// TIA Portal V19 export
FUNCTION "FC_001_Diagnostic" : Void   // FC12, LAD
{ S7_Optimized_Access := 'TRUE' }
// stored: SetENOAutomatically false
   VAR_IN_OUT
      Diagnostic7 : "DiagnosticMainCabinet";
      Diagnostic10 : "DiagnosticMainCabinet";
   END_VAR
BEGIN

REGION Network 1 (SCL)
   //************************************************************
   //===Author: Mateusz Połojko
   //-----Linkedin: https://pl.linkedin.com/in/mateusz-po%C5%82ojko-52a3541b1
   //-----Github: https://github.com/Bhazel95
   //===Description:
   //-----Diagnostic of hardware components
   //===Customer:
   //-----Apator Powogaz S.A.
   //************************************************************
END_REGION

REGION Network 2 (SCL)
   //Transporter 7A & 7B
   #Diagnostic7.ET_200SP.HeadModule_0.LADDR:= "IO_device_1~Head";
   #Diagnostic7.ET_200SP.HeadModule_0.Mode := 1;

   #Diagnostic7.ET_200SP.BusAdapter_1.LADDR := "IO_device_1~BusAdapter-Send_1xFC_1";
   #Diagnostic7.ET_200SP.BusAdapter_1.Mode := 1;

   #Diagnostic7.ET_200SP.InputSafety_2.LADDR := "IO_device_1~F-DI_8x24VDC_HF_1" ;
   #Diagnostic7.ET_200SP.InputSafety_2.Mode := 1;

   #Diagnostic7.ET_200SP.InputSafety_3.LADDR := "IO_device_1~F-DI_8x24VDC_HF_2";
   #Diagnostic7.ET_200SP.InputSafety_3.Mode := 1;

   #Diagnostic7.ET_200SP.InputSafety_4.LADDR := "IO_device_1~F-DI_8x24VDC_HF_3";
   #Diagnostic7.ET_200SP.InputSafety_4.Mode := 1;

   #Diagnostic7.ET_200SP.InputSafety_5.LADDR := "IO_device_1~F-DI_8x24VDC_HF_5";
   #Diagnostic7.ET_200SP.InputSafety_5.Mode := 1;

   #Diagnostic7.ET_200SP.InputSafety_6.LADDR := "IO_device_1~F-DI_8x24VDC_HF_4";
   #Diagnostic7.ET_200SP.InputSafety_6.Mode := 1;

   #Diagnostic7.ET_200SP.OutputSafety_7.LADDR := "IO_device_1~F-DQ_8x24VDC_0_5A_PP_HF_1";
   #Diagnostic7.ET_200SP.OutputSafety_7.Mode := 1;

   #Diagnostic7.ET_200SP.RelaySafety_9.LADDR := "IO_device_1~F-RQ_1x24__48VDC_24__230VAC_5A_1";
   #Diagnostic7.ET_200SP.RelaySafety_9.Mode := 1;

   #Diagnostic7.ET_200SP.RelaySafety_10.LADDR := "IO_device_1~F-RQ_1x24__48VDC_24__230VAC_5A_2";
   #Diagnostic7.ET_200SP.RelaySafety_10.Mode := 1;

   #Diagnostic7.ET_200SP.InputsDigital_11.LADDR := "IO_device_1~DI_16x24VDC_ST_1";
   #Diagnostic7.ET_200SP.InputsDigital_11.Mode := 1;

   #Diagnostic7.ET_200SP.InputsDigital_12.LADDR := "IO_device_1~DI_16x24VDC_ST_2";
   #Diagnostic7.ET_200SP.InputsDigital_12.Mode := 1;

   #Diagnostic7.ET_200SP.InputsDigital_13.LADDR := "IO_device_1~DI_16x24VDC_ST_3";
   #Diagnostic7.ET_200SP.InputsDigital_13.Mode := 1;

   #Diagnostic7.ET_200SP.InputAnalog_14.LADDR := "IO_device_1~AI_2xI_2-_4-wire_ST_1";
   #Diagnostic7.ET_200SP.InputAnalog_14.Mode := 1;

   #Diagnostic7.ET_200SP.OutputDigital_15.LADDR := "IO_device_1~DQ_16x24VDC_0_5A_ST_1";
   #Diagnostic7.ET_200SP.OutputDigital_15.Mode := 1;

   #Diagnostic7.ET_200SP.OutputDigital_16.LADDR := "IO_device_1~DQ_16x24VDC_0_5A_ST_2";
   #Diagnostic7.ET_200SP.OutputDigital_16.Mode := 1;

   #Diagnostic7.ET_200SP.OutputDigital_17.LADDR := "IO_device_1~DQ_16x24VDC_0_5A_ST_3";
   #Diagnostic7.ET_200SP.OutputDigital_17.Mode := 1;

   #Diagnostic7.ET_200SP.OutputDigital_18.LADDR := "IO_device_1~DQ_16x24VDC_0_5A_ST_4";
   #Diagnostic7.ET_200SP.OutputDigital_18.Mode := 1;

   #Diagnostic7.ET_200SP.OutputAnalog_19.LADDR := "IO_device_1~AQ_2xI_ST_1";
   #Diagnostic7.ET_200SP.OutputAnalog_19.Mode := 1;

   #Diagnostic7.ET_200SP.ET_200AL_1.LADDR := "IO_device_1~DI_8x24VDC_8xM8_1";
   #Diagnostic7.ET_200SP.ET_200AL_1.Mode := 1;

   #Diagnostic7.ET_200SP.ET_200AL_2.LADDR := "IO_device_1~DI_8x24VDC_8xM8_2";
   #Diagnostic7.ET_200SP.ET_200AL_2.Mode := 1;


   #Diagnostic7.SinamicG120_1.LADDR := "G120_CU250S_2_PN_VECTOR_7A~PROFINET_interface~IODevice";
   #Diagnostic7.SinamicG120_1.Mode := 1;

   #Diagnostic7.SinamicG120_1.LADDR := "G120_CU250S_2_PN_VECTOR_7B~PROFINET_interface~IODevice";
   #Diagnostic7.SinamicG120_1.Mode := 1;
END_REGION

REGION Network 3 (SCL)
   //Transporter 10A & 10B
   #Diagnostic10.ET_200SP.HeadModule_0.LADDR := "IO_device_2~Head";
   #Diagnostic10.ET_200SP.HeadModule_0.Mode := 1;

   #Diagnostic10.ET_200SP.BusAdapter_1.LADDR := "IO_device_2~BusAdapter-Send_1xFC_1";
   #Diagnostic10.ET_200SP.BusAdapter_1.Mode := 1;

   #Diagnostic10.ET_200SP.InputSafety_2.LADDR := "IO_device_2~F-DI_8x24VDC_HF_1";
   #Diagnostic10.ET_200SP.InputSafety_2.Mode := 1;

   #Diagnostic10.ET_200SP.InputSafety_3.LADDR := "IO_device_2~F-DI_8x24VDC_HF_2";
   #Diagnostic10.ET_200SP.InputSafety_3.Mode := 1;

   #Diagnostic10.ET_200SP.InputSafety_4.LADDR := "IO_device_2~F-DI_8x24VDC_HF_3";
   #Diagnostic10.ET_200SP.InputSafety_4.Mode := 1;

   #Diagnostic10.ET_200SP.InputSafety_5.LADDR := "IO_device_2~F-DI_8x24VDC_HF_4";
   #Diagnostic10.ET_200SP.InputSafety_5.Mode := 1;

   #Diagnostic10.ET_200SP.InputSafety_6.LADDR := "IO_device_2~F-DI_8x24VDC_HF_5";
   #Diagnostic10.ET_200SP.InputSafety_6.Mode := 1;

   #Diagnostic10.ET_200SP.OutputSafety_7.LADDR := "IO_device_2~F-DQ_8x24VDC_0_5A_PP_HF_1";
   #Diagnostic10.ET_200SP.OutputSafety_7.Mode := 1;

   #Diagnostic10.ET_200SP.RelaySafety_9.LADDR := "IO_device_2~F-RQ_1x24__48VDC_24__230VAC_5A_1";
   #Diagnostic10.ET_200SP.RelaySafety_9.Mode := 1;

   #Diagnostic10.ET_200SP.RelaySafety_10.LADDR := "IO_device_2~F-RQ_1x24__48VDC_24__230VAC_5A_2";
   #Diagnostic10.ET_200SP.RelaySafety_10.Mode := 1;

   #Diagnostic10.ET_200SP.InputsDigital_11.LADDR := "IO_device_2~DI_16x24VDC_ST_1";
   #Diagnostic10.ET_200SP.InputsDigital_11.Mode := 1;

   #Diagnostic10.ET_200SP.InputsDigital_12.LADDR := "IO_device_2~DI_16x24VDC_ST_2";
   #Diagnostic10.ET_200SP.InputsDigital_12.Mode := 1;

   #Diagnostic10.ET_200SP.InputsDigital_13.LADDR := "IO_device_2~DI_16x24VDC_ST_3";
   #Diagnostic10.ET_200SP.InputsDigital_13.Mode := 1;

   #Diagnostic10.ET_200SP.InputAnalog_14.LADDR := "IO_device_2~AI_2xI_2-_4-wire_ST_1";
   #Diagnostic10.ET_200SP.InputAnalog_14.Mode := 1;

   #Diagnostic10.ET_200SP.OutputDigital_15.LADDR := "IO_device_2~DQ_16x24VDC_0_5A_ST_1";
   #Diagnostic10.ET_200SP.OutputDigital_15.Mode := 1;

   #Diagnostic10.ET_200SP.OutputDigital_16.LADDR := "IO_device_2~DQ_16x24VDC_0_5A_ST_2";
   #Diagnostic10.ET_200SP.OutputDigital_16.Mode := 1;

   #Diagnostic10.ET_200SP.OutputDigital_17.LADDR := "IO_device_2~DQ_16x24VDC_0_5A_ST_3";
   #Diagnostic10.ET_200SP.OutputDigital_17.Mode := 1;

   #Diagnostic10.ET_200SP.OutputDigital_18.LADDR := "IO_device_2~DQ_16x24VDC_0_5A_ST_4";
   #Diagnostic10.ET_200SP.OutputDigital_18.Mode := 1;

   #Diagnostic10.ET_200SP.OutputAnalog_19.LADDR := "IO_device_2~AQ_2xI_ST_1";
   #Diagnostic10.ET_200SP.OutputAnalog_19.Mode := 1;

   #Diagnostic10.ET_200SP.ET_200AL_1.LADDR := "IO_device_2~DI_8x24VDC_8xM8_1";
   #Diagnostic10.ET_200SP.ET_200AL_1.Mode := 1;

   #Diagnostic10.ET_200SP.ET_200AL_2.LADDR := "IO_device_2~DI_8x24VDC_8xM8_2";
   #Diagnostic10.ET_200SP.ET_200AL_2.Mode := 1;


   #Diagnostic10.SinamicG120_1.LADDR := "G120_CU250S_2_PN_VECTOR_10A~PROFINET_interface~IODevice";
   #Diagnostic10.SinamicG120_1.Mode := 1;
END_REGION

REGION Network 4
   // ET 200SP - MODUL GLOWNY 7
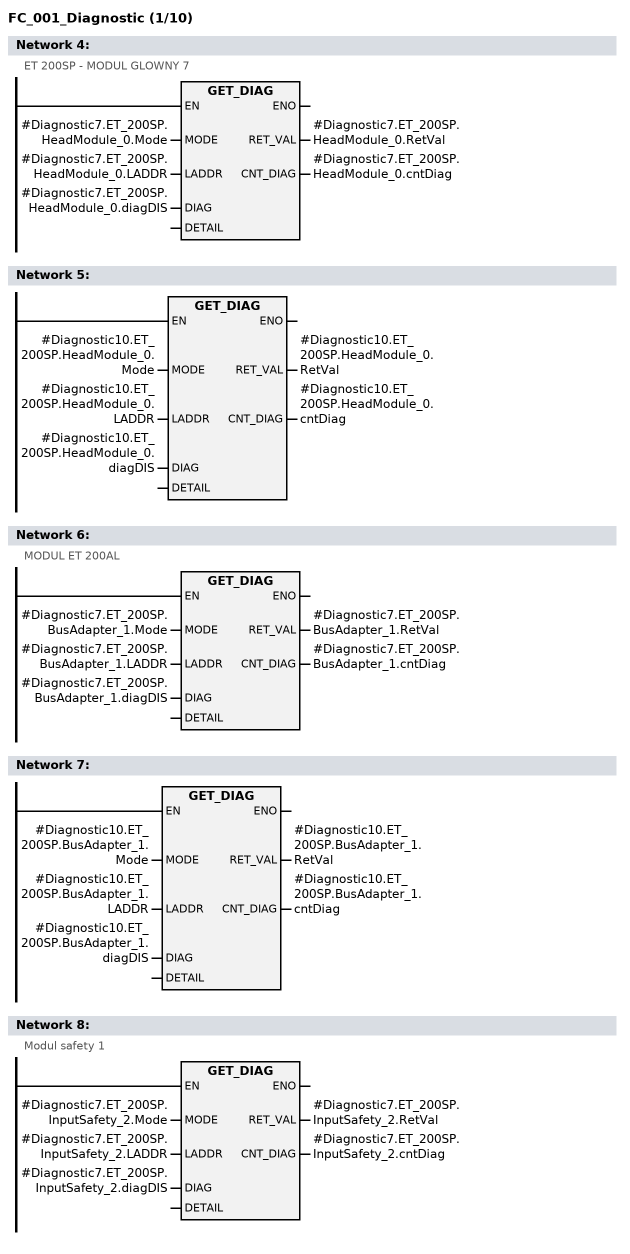
   RUNG wire#powerrail
      GET_DIAG(MODE := #Diagnostic7.ET_200SP.HeadModule_0.Mode, LADDR := #Diagnostic7.ET_200SP.HeadModule_0.LADDR, DIAG := #Diagnostic7.ET_200SP.HeadModule_0.diagDIS, DETAIL :=, RET_VAL => #Diagnostic7.ET_200SP.HeadModule_0.RetVal, CNT_DIAG => #Diagnostic7.ET_200SP.HeadModule_0.cntDiag)
   END_RUNG
   // the same network as SCL:
   #Diagnostic7.ET_200SP.HeadModule_0.RetVal := GET_DIAG(MODE := #Diagnostic7.ET_200SP.HeadModule_0.Mode,
                           LADDR := #Diagnostic7.ET_200SP.HeadModule_0.LADDR,
                           DIAG := #Diagnostic7.ET_200SP.HeadModule_0.diagDIS,
                           CNT_DIAG => #Diagnostic7.ET_200SP.HeadModule_0.cntDiag);
END_REGION

REGION Network 5
   RUNG wire#powerrail
      GET_DIAG(MODE := #Diagnostic10.ET_200SP.HeadModule_0.Mode, LADDR := #Diagnostic10.ET_200SP.HeadModule_0.LADDR, DIAG := #Diagnostic10.ET_200SP.HeadModule_0.diagDIS, DETAIL :=, RET_VAL => #Diagnostic10.ET_200SP.HeadModule_0.RetVal, CNT_DIAG => #Diagnostic10.ET_200SP.HeadModule_0.cntDiag)
   END_RUNG
   // the same network as SCL:
   #Diagnostic10.ET_200SP.HeadModule_0.RetVal := GET_DIAG(MODE := #Diagnostic10.ET_200SP.HeadModule_0.Mode,
                           LADDR := #Diagnostic10.ET_200SP.HeadModule_0.LADDR,
                           DIAG := #Diagnostic10.ET_200SP.HeadModule_0.diagDIS,
                           CNT_DIAG => #Diagnostic10.ET_200SP.HeadModule_0.cntDiag);
END_REGION

REGION Network 6
   // MODUL ET 200AL
   RUNG wire#powerrail
      GET_DIAG(MODE := #Diagnostic7.ET_200SP.BusAdapter_1.Mode, LADDR := #Diagnostic7.ET_200SP.BusAdapter_1.LADDR, DIAG := #Diagnostic7.ET_200SP.BusAdapter_1.diagDIS, DETAIL :=, RET_VAL => #Diagnostic7.ET_200SP.BusAdapter_1.RetVal, CNT_DIAG => #Diagnostic7.ET_200SP.BusAdapter_1.cntDiag)
   END_RUNG
   // the same network as SCL:
   #Diagnostic7.ET_200SP.BusAdapter_1.RetVal := GET_DIAG(MODE := #Diagnostic7.ET_200SP.BusAdapter_1.Mode,
                           LADDR := #Diagnostic7.ET_200SP.BusAdapter_1.LADDR,
                           DIAG := #Diagnostic7.ET_200SP.BusAdapter_1.diagDIS,
                           CNT_DIAG => #Diagnostic7.ET_200SP.BusAdapter_1.cntDiag);
END_REGION

REGION Network 7
   RUNG wire#powerrail
      GET_DIAG(MODE := #Diagnostic10.ET_200SP.BusAdapter_1.Mode, LADDR := #Diagnostic10.ET_200SP.BusAdapter_1.LADDR, DIAG := #Diagnostic10.ET_200SP.BusAdapter_1.diagDIS, DETAIL :=, RET_VAL => #Diagnostic10.ET_200SP.BusAdapter_1.RetVal, CNT_DIAG => #Diagnostic10.ET_200SP.BusAdapter_1.cntDiag)
   END_RUNG
   // the same network as SCL:
   #Diagnostic10.ET_200SP.BusAdapter_1.RetVal := GET_DIAG(MODE := #Diagnostic10.ET_200SP.BusAdapter_1.Mode,
                           LADDR := #Diagnostic10.ET_200SP.BusAdapter_1.LADDR,
                           DIAG := #Diagnostic10.ET_200SP.BusAdapter_1.diagDIS,
                           CNT_DIAG => #Diagnostic10.ET_200SP.BusAdapter_1.cntDiag);
END_REGION

REGION Network 8
   // Modul safety 1
   RUNG wire#powerrail
      GET_DIAG(MODE := #Diagnostic7.ET_200SP.InputSafety_2.Mode, LADDR := #Diagnostic7.ET_200SP.InputSafety_2.LADDR, DIAG := #Diagnostic7.ET_200SP.InputSafety_2.diagDIS, DETAIL :=, RET_VAL => #Diagnostic7.ET_200SP.InputSafety_2.RetVal, CNT_DIAG => #Diagnostic7.ET_200SP.InputSafety_2.cntDiag)
   END_RUNG
   // the same network as SCL:
   #Diagnostic7.ET_200SP.InputSafety_2.RetVal := GET_DIAG(MODE := #Diagnostic7.ET_200SP.InputSafety_2.Mode,
                           LADDR := #Diagnostic7.ET_200SP.InputSafety_2.LADDR,
                           DIAG := #Diagnostic7.ET_200SP.InputSafety_2.diagDIS,
                           CNT_DIAG => #Diagnostic7.ET_200SP.InputSafety_2.cntDiag);
END_REGION

REGION Network 9
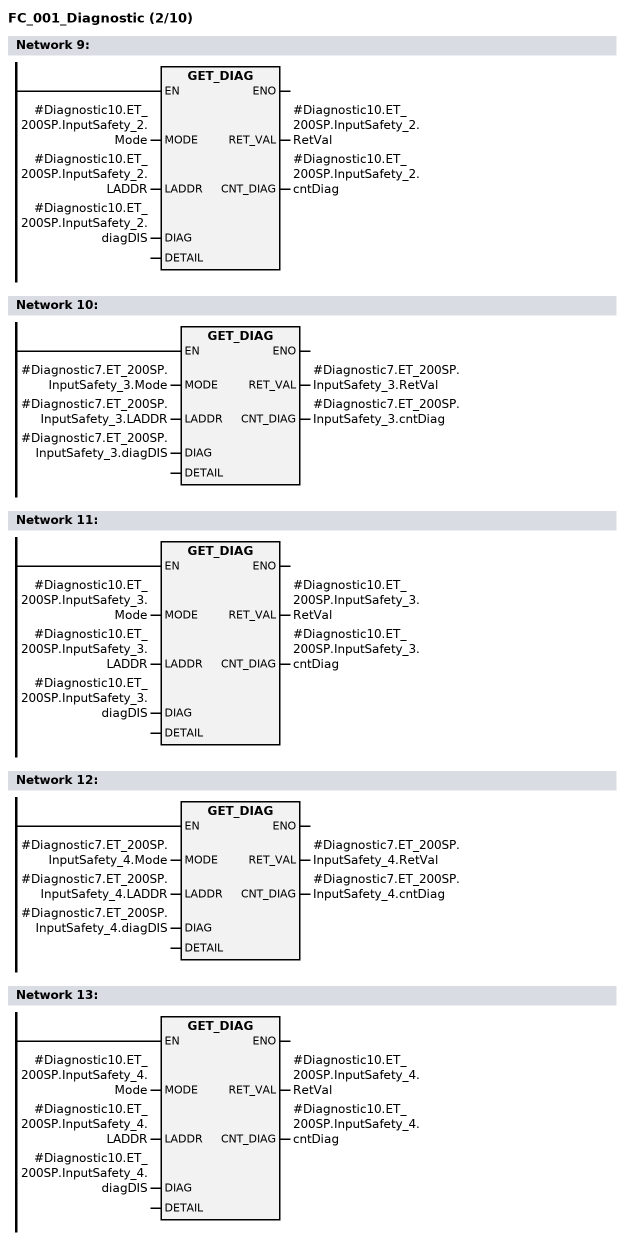
   RUNG wire#powerrail
      GET_DIAG(MODE := #Diagnostic10.ET_200SP.InputSafety_2.Mode, LADDR := #Diagnostic10.ET_200SP.InputSafety_2.LADDR, DIAG := #Diagnostic10.ET_200SP.InputSafety_2.diagDIS, DETAIL :=, RET_VAL => #Diagnostic10.ET_200SP.InputSafety_2.RetVal, CNT_DIAG => #Diagnostic10.ET_200SP.InputSafety_2.cntDiag)
   END_RUNG
   // the same network as SCL:
   #Diagnostic10.ET_200SP.InputSafety_2.RetVal := GET_DIAG(MODE := #Diagnostic10.ET_200SP.InputSafety_2.Mode,
                           LADDR := #Diagnostic10.ET_200SP.InputSafety_2.LADDR,
                           DIAG := #Diagnostic10.ET_200SP.InputSafety_2.diagDIS,
                           CNT_DIAG => #Diagnostic10.ET_200SP.InputSafety_2.cntDiag);
END_REGION

REGION Network 10
   RUNG wire#powerrail
      GET_DIAG(MODE := #Diagnostic7.ET_200SP.InputSafety_3.Mode, LADDR := #Diagnostic7.ET_200SP.InputSafety_3.LADDR, DIAG := #Diagnostic7.ET_200SP.InputSafety_3.diagDIS, DETAIL :=, RET_VAL => #Diagnostic7.ET_200SP.InputSafety_3.RetVal, CNT_DIAG => #Diagnostic7.ET_200SP.InputSafety_3.cntDiag)
   END_RUNG
   // the same network as SCL:
   #Diagnostic7.ET_200SP.InputSafety_3.RetVal := GET_DIAG(MODE := #Diagnostic7.ET_200SP.InputSafety_3.Mode,
                           LADDR := #Diagnostic7.ET_200SP.InputSafety_3.LADDR,
                           DIAG := #Diagnostic7.ET_200SP.InputSafety_3.diagDIS,
                           CNT_DIAG => #Diagnostic7.ET_200SP.InputSafety_3.cntDiag);
END_REGION

REGION Network 11
   RUNG wire#powerrail
      GET_DIAG(MODE := #Diagnostic10.ET_200SP.InputSafety_3.Mode, LADDR := #Diagnostic10.ET_200SP.InputSafety_3.LADDR, DIAG := #Diagnostic10.ET_200SP.InputSafety_3.diagDIS, DETAIL :=, RET_VAL => #Diagnostic10.ET_200SP.InputSafety_3.RetVal, CNT_DIAG => #Diagnostic10.ET_200SP.InputSafety_3.cntDiag)
   END_RUNG
   // the same network as SCL:
   #Diagnostic10.ET_200SP.InputSafety_3.RetVal := GET_DIAG(MODE := #Diagnostic10.ET_200SP.InputSafety_3.Mode,
                           LADDR := #Diagnostic10.ET_200SP.InputSafety_3.LADDR,
                           DIAG := #Diagnostic10.ET_200SP.InputSafety_3.diagDIS,
                           CNT_DIAG => #Diagnostic10.ET_200SP.InputSafety_3.cntDiag);
END_REGION

REGION Network 12
   RUNG wire#powerrail
      GET_DIAG(MODE := #Diagnostic7.ET_200SP.InputSafety_4.Mode, LADDR := #Diagnostic7.ET_200SP.InputSafety_4.LADDR, DIAG := #Diagnostic7.ET_200SP.InputSafety_4.diagDIS, DETAIL :=, RET_VAL => #Diagnostic7.ET_200SP.InputSafety_4.RetVal, CNT_DIAG => #Diagnostic7.ET_200SP.InputSafety_4.cntDiag)
   END_RUNG
   // the same network as SCL:
   #Diagnostic7.ET_200SP.InputSafety_4.RetVal := GET_DIAG(MODE := #Diagnostic7.ET_200SP.InputSafety_4.Mode,
                           LADDR := #Diagnostic7.ET_200SP.InputSafety_4.LADDR,
                           DIAG := #Diagnostic7.ET_200SP.InputSafety_4.diagDIS,
                           CNT_DIAG => #Diagnostic7.ET_200SP.InputSafety_4.cntDiag);
END_REGION

REGION Network 13
   RUNG wire#powerrail
      GET_DIAG(MODE := #Diagnostic10.ET_200SP.InputSafety_4.Mode, LADDR := #Diagnostic10.ET_200SP.InputSafety_4.LADDR, DIAG := #Diagnostic10.ET_200SP.InputSafety_4.diagDIS, DETAIL :=, RET_VAL => #Diagnostic10.ET_200SP.InputSafety_4.RetVal, CNT_DIAG => #Diagnostic10.ET_200SP.InputSafety_4.cntDiag)
   END_RUNG
   // the same network as SCL:
   #Diagnostic10.ET_200SP.InputSafety_4.RetVal := GET_DIAG(MODE := #Diagnostic10.ET_200SP.InputSafety_4.Mode,
                           LADDR := #Diagnostic10.ET_200SP.InputSafety_4.LADDR,
                           DIAG := #Diagnostic10.ET_200SP.InputSafety_4.diagDIS,
                           CNT_DIAG => #Diagnostic10.ET_200SP.InputSafety_4.cntDiag);
END_REGION

REGION Network 14
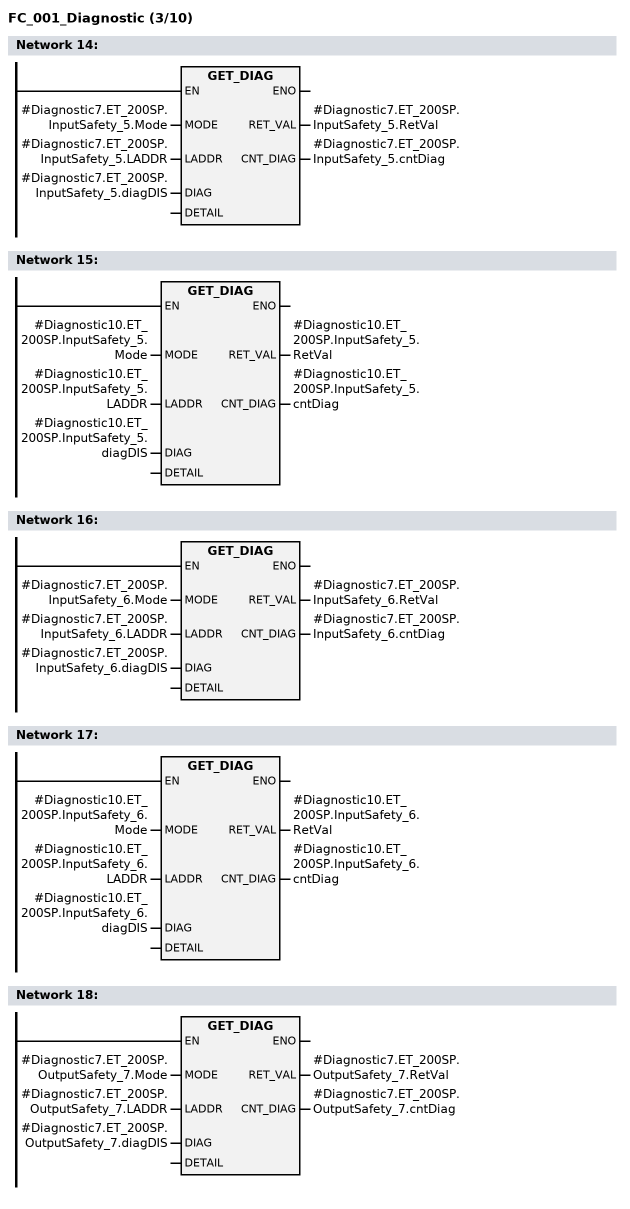
   RUNG wire#powerrail
      GET_DIAG(MODE := #Diagnostic7.ET_200SP.InputSafety_5.Mode, LADDR := #Diagnostic7.ET_200SP.InputSafety_5.LADDR, DIAG := #Diagnostic7.ET_200SP.InputSafety_5.diagDIS, DETAIL :=, RET_VAL => #Diagnostic7.ET_200SP.InputSafety_5.RetVal, CNT_DIAG => #Diagnostic7.ET_200SP.InputSafety_5.cntDiag)
   END_RUNG
   // the same network as SCL:
   #Diagnostic7.ET_200SP.InputSafety_5.RetVal := GET_DIAG(MODE := #Diagnostic7.ET_200SP.InputSafety_5.Mode,
                           LADDR := #Diagnostic7.ET_200SP.InputSafety_5.LADDR,
                           DIAG := #Diagnostic7.ET_200SP.InputSafety_5.diagDIS,
                           CNT_DIAG => #Diagnostic7.ET_200SP.InputSafety_5.cntDiag);
END_REGION

REGION Network 15
   RUNG wire#powerrail
      GET_DIAG(MODE := #Diagnostic10.ET_200SP.InputSafety_5.Mode, LADDR := #Diagnostic10.ET_200SP.InputSafety_5.LADDR, DIAG := #Diagnostic10.ET_200SP.InputSafety_5.diagDIS, DETAIL :=, RET_VAL => #Diagnostic10.ET_200SP.InputSafety_5.RetVal, CNT_DIAG => #Diagnostic10.ET_200SP.InputSafety_5.cntDiag)
   END_RUNG
   // the same network as SCL:
   #Diagnostic10.ET_200SP.InputSafety_5.RetVal := GET_DIAG(MODE := #Diagnostic10.ET_200SP.InputSafety_5.Mode,
                           LADDR := #Diagnostic10.ET_200SP.InputSafety_5.LADDR,
                           DIAG := #Diagnostic10.ET_200SP.InputSafety_5.diagDIS,
                           CNT_DIAG => #Diagnostic10.ET_200SP.InputSafety_5.cntDiag);
END_REGION

REGION Network 16
   RUNG wire#powerrail
      GET_DIAG(MODE := #Diagnostic7.ET_200SP.InputSafety_6.Mode, LADDR := #Diagnostic7.ET_200SP.InputSafety_6.LADDR, DIAG := #Diagnostic7.ET_200SP.InputSafety_6.diagDIS, DETAIL :=, RET_VAL => #Diagnostic7.ET_200SP.InputSafety_6.RetVal, CNT_DIAG => #Diagnostic7.ET_200SP.InputSafety_6.cntDiag)
   END_RUNG
   // the same network as SCL:
   #Diagnostic7.ET_200SP.InputSafety_6.RetVal := GET_DIAG(MODE := #Diagnostic7.ET_200SP.InputSafety_6.Mode,
                           LADDR := #Diagnostic7.ET_200SP.InputSafety_6.LADDR,
                           DIAG := #Diagnostic7.ET_200SP.InputSafety_6.diagDIS,
                           CNT_DIAG => #Diagnostic7.ET_200SP.InputSafety_6.cntDiag);
END_REGION

REGION Network 17
   RUNG wire#powerrail
      GET_DIAG(MODE := #Diagnostic10.ET_200SP.InputSafety_6.Mode, LADDR := #Diagnostic10.ET_200SP.InputSafety_6.LADDR, DIAG := #Diagnostic10.ET_200SP.InputSafety_6.diagDIS, DETAIL :=, RET_VAL => #Diagnostic10.ET_200SP.InputSafety_6.RetVal, CNT_DIAG => #Diagnostic10.ET_200SP.InputSafety_6.cntDiag)
   END_RUNG
   // the same network as SCL:
   #Diagnostic10.ET_200SP.InputSafety_6.RetVal := GET_DIAG(MODE := #Diagnostic10.ET_200SP.InputSafety_6.Mode,
                           LADDR := #Diagnostic10.ET_200SP.InputSafety_6.LADDR,
                           DIAG := #Diagnostic10.ET_200SP.InputSafety_6.diagDIS,
                           CNT_DIAG => #Diagnostic10.ET_200SP.InputSafety_6.cntDiag);
END_REGION

REGION Network 18
   RUNG wire#powerrail
      GET_DIAG(MODE := #Diagnostic7.ET_200SP.OutputSafety_7.Mode, LADDR := #Diagnostic7.ET_200SP.OutputSafety_7.LADDR, DIAG := #Diagnostic7.ET_200SP.OutputSafety_7.diagDIS, DETAIL :=, RET_VAL => #Diagnostic7.ET_200SP.OutputSafety_7.RetVal, CNT_DIAG => #Diagnostic7.ET_200SP.OutputSafety_7.cntDiag)
   END_RUNG
   // the same network as SCL:
   #Diagnostic7.ET_200SP.OutputSafety_7.RetVal := GET_DIAG(MODE := #Diagnostic7.ET_200SP.OutputSafety_7.Mode,
                           LADDR := #Diagnostic7.ET_200SP.OutputSafety_7.LADDR,
                           DIAG := #Diagnostic7.ET_200SP.OutputSafety_7.diagDIS,
                           CNT_DIAG => #Diagnostic7.ET_200SP.OutputSafety_7.cntDiag);
END_REGION

REGION Network 19
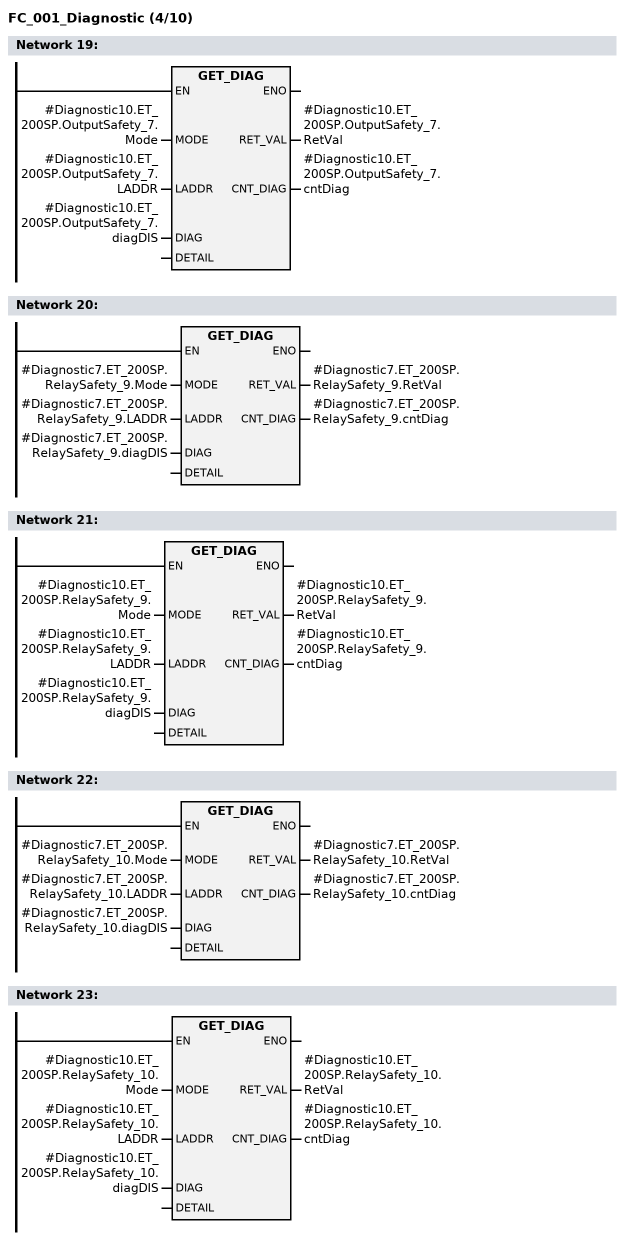
   RUNG wire#powerrail
      GET_DIAG(MODE := #Diagnostic10.ET_200SP.OutputSafety_7.Mode, LADDR := #Diagnostic10.ET_200SP.OutputSafety_7.LADDR, DIAG := #Diagnostic10.ET_200SP.OutputSafety_7.diagDIS, DETAIL :=, RET_VAL => #Diagnostic10.ET_200SP.OutputSafety_7.RetVal, CNT_DIAG => #Diagnostic10.ET_200SP.OutputSafety_7.cntDiag)
   END_RUNG
   // the same network as SCL:
   #Diagnostic10.ET_200SP.OutputSafety_7.RetVal := GET_DIAG(MODE := #Diagnostic10.ET_200SP.OutputSafety_7.Mode,
                           LADDR := #Diagnostic10.ET_200SP.OutputSafety_7.LADDR,
                           DIAG := #Diagnostic10.ET_200SP.OutputSafety_7.diagDIS,
                           CNT_DIAG => #Diagnostic10.ET_200SP.OutputSafety_7.cntDiag);
END_REGION

REGION Network 20
   RUNG wire#powerrail
      GET_DIAG(MODE := #Diagnostic7.ET_200SP.RelaySafety_9.Mode, LADDR := #Diagnostic7.ET_200SP.RelaySafety_9.LADDR, DIAG := #Diagnostic7.ET_200SP.RelaySafety_9.diagDIS, DETAIL :=, RET_VAL => #Diagnostic7.ET_200SP.RelaySafety_9.RetVal, CNT_DIAG => #Diagnostic7.ET_200SP.RelaySafety_9.cntDiag)
   END_RUNG
   // the same network as SCL:
   #Diagnostic7.ET_200SP.RelaySafety_9.RetVal := GET_DIAG(MODE := #Diagnostic7.ET_200SP.RelaySafety_9.Mode,
                           LADDR := #Diagnostic7.ET_200SP.RelaySafety_9.LADDR,
                           DIAG := #Diagnostic7.ET_200SP.RelaySafety_9.diagDIS,
                           CNT_DIAG => #Diagnostic7.ET_200SP.RelaySafety_9.cntDiag);
END_REGION

REGION Network 21
   RUNG wire#powerrail
      GET_DIAG(MODE := #Diagnostic10.ET_200SP.RelaySafety_9.Mode, LADDR := #Diagnostic10.ET_200SP.RelaySafety_9.LADDR, DIAG := #Diagnostic10.ET_200SP.RelaySafety_9.diagDIS, DETAIL :=, RET_VAL => #Diagnostic10.ET_200SP.RelaySafety_9.RetVal, CNT_DIAG => #Diagnostic10.ET_200SP.RelaySafety_9.cntDiag)
   END_RUNG
   // the same network as SCL:
   #Diagnostic10.ET_200SP.RelaySafety_9.RetVal := GET_DIAG(MODE := #Diagnostic10.ET_200SP.RelaySafety_9.Mode,
                           LADDR := #Diagnostic10.ET_200SP.RelaySafety_9.LADDR,
                           DIAG := #Diagnostic10.ET_200SP.RelaySafety_9.diagDIS,
                           CNT_DIAG => #Diagnostic10.ET_200SP.RelaySafety_9.cntDiag);
END_REGION

REGION Network 22
   RUNG wire#powerrail
      GET_DIAG(MODE := #Diagnostic7.ET_200SP.RelaySafety_10.Mode, LADDR := #Diagnostic7.ET_200SP.RelaySafety_10.LADDR, DIAG := #Diagnostic7.ET_200SP.RelaySafety_10.diagDIS, DETAIL :=, RET_VAL => #Diagnostic7.ET_200SP.RelaySafety_10.RetVal, CNT_DIAG => #Diagnostic7.ET_200SP.RelaySafety_10.cntDiag)
   END_RUNG
   // the same network as SCL:
   #Diagnostic7.ET_200SP.RelaySafety_10.RetVal := GET_DIAG(MODE := #Diagnostic7.ET_200SP.RelaySafety_10.Mode,
                           LADDR := #Diagnostic7.ET_200SP.RelaySafety_10.LADDR,
                           DIAG := #Diagnostic7.ET_200SP.RelaySafety_10.diagDIS,
                           CNT_DIAG => #Diagnostic7.ET_200SP.RelaySafety_10.cntDiag);
END_REGION

REGION Network 23
   RUNG wire#powerrail
      GET_DIAG(MODE := #Diagnostic10.ET_200SP.RelaySafety_10.Mode, LADDR := #Diagnostic10.ET_200SP.RelaySafety_10.LADDR, DIAG := #Diagnostic10.ET_200SP.RelaySafety_10.diagDIS, DETAIL :=, RET_VAL => #Diagnostic10.ET_200SP.RelaySafety_10.RetVal, CNT_DIAG => #Diagnostic10.ET_200SP.RelaySafety_10.cntDiag)
   END_RUNG
   // the same network as SCL:
   #Diagnostic10.ET_200SP.RelaySafety_10.RetVal := GET_DIAG(MODE := #Diagnostic10.ET_200SP.RelaySafety_10.Mode,
                           LADDR := #Diagnostic10.ET_200SP.RelaySafety_10.LADDR,
                           DIAG := #Diagnostic10.ET_200SP.RelaySafety_10.diagDIS,
                           CNT_DIAG => #Diagnostic10.ET_200SP.RelaySafety_10.cntDiag);
END_REGION

REGION Network 24
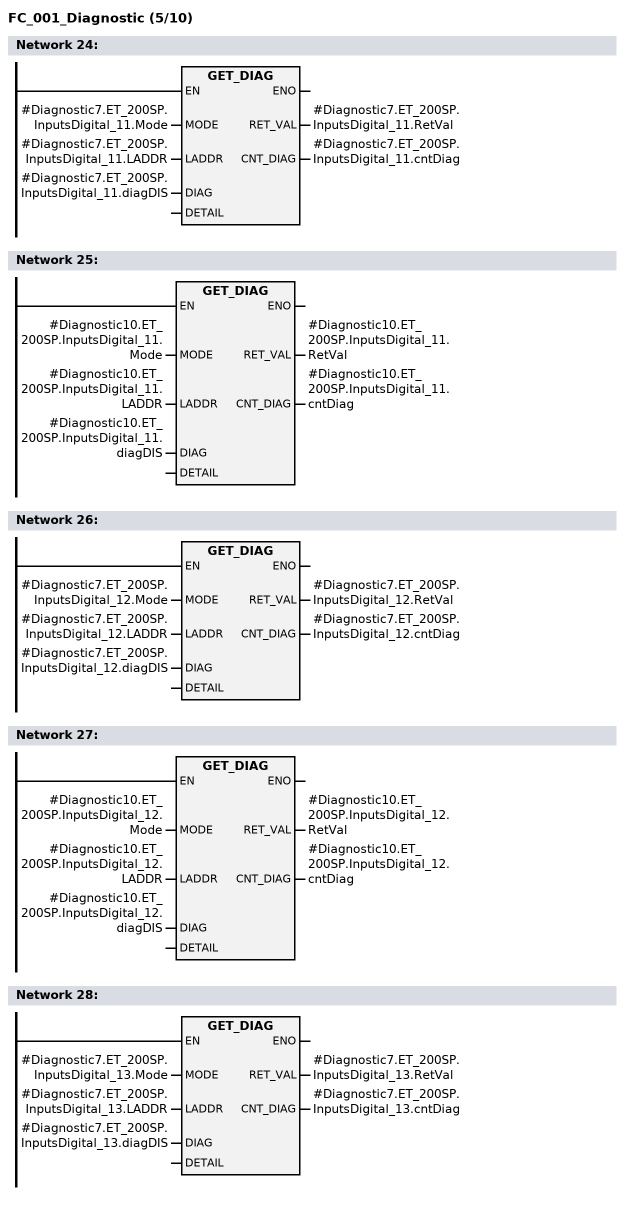
   RUNG wire#powerrail
      GET_DIAG(MODE := #Diagnostic7.ET_200SP.InputsDigital_11.Mode, LADDR := #Diagnostic7.ET_200SP.InputsDigital_11.LADDR, DIAG := #Diagnostic7.ET_200SP.InputsDigital_11.diagDIS, DETAIL :=, RET_VAL => #Diagnostic7.ET_200SP.InputsDigital_11.RetVal, CNT_DIAG => #Diagnostic7.ET_200SP.InputsDigital_11.cntDiag)
   END_RUNG
   // the same network as SCL:
   #Diagnostic7.ET_200SP.InputsDigital_11.RetVal := GET_DIAG(MODE := #Diagnostic7.ET_200SP.InputsDigital_11.Mode,
                           LADDR := #Diagnostic7.ET_200SP.InputsDigital_11.LADDR,
                           DIAG := #Diagnostic7.ET_200SP.InputsDigital_11.diagDIS,
                           CNT_DIAG => #Diagnostic7.ET_200SP.InputsDigital_11.cntDiag);
END_REGION

REGION Network 25
   RUNG wire#powerrail
      GET_DIAG(MODE := #Diagnostic10.ET_200SP.InputsDigital_11.Mode, LADDR := #Diagnostic10.ET_200SP.InputsDigital_11.LADDR, DIAG := #Diagnostic10.ET_200SP.InputsDigital_11.diagDIS, DETAIL :=, RET_VAL => #Diagnostic10.ET_200SP.InputsDigital_11.RetVal, CNT_DIAG => #Diagnostic10.ET_200SP.InputsDigital_11.cntDiag)
   END_RUNG
   // the same network as SCL:
   #Diagnostic10.ET_200SP.InputsDigital_11.RetVal := GET_DIAG(MODE := #Diagnostic10.ET_200SP.InputsDigital_11.Mode,
                           LADDR := #Diagnostic10.ET_200SP.InputsDigital_11.LADDR,
                           DIAG := #Diagnostic10.ET_200SP.InputsDigital_11.diagDIS,
                           CNT_DIAG => #Diagnostic10.ET_200SP.InputsDigital_11.cntDiag);
END_REGION

REGION Network 26
   RUNG wire#powerrail
      GET_DIAG(MODE := #Diagnostic7.ET_200SP.InputsDigital_12.Mode, LADDR := #Diagnostic7.ET_200SP.InputsDigital_12.LADDR, DIAG := #Diagnostic7.ET_200SP.InputsDigital_12.diagDIS, DETAIL :=, RET_VAL => #Diagnostic7.ET_200SP.InputsDigital_12.RetVal, CNT_DIAG => #Diagnostic7.ET_200SP.InputsDigital_12.cntDiag)
   END_RUNG
   // the same network as SCL:
   #Diagnostic7.ET_200SP.InputsDigital_12.RetVal := GET_DIAG(MODE := #Diagnostic7.ET_200SP.InputsDigital_12.Mode,
                           LADDR := #Diagnostic7.ET_200SP.InputsDigital_12.LADDR,
                           DIAG := #Diagnostic7.ET_200SP.InputsDigital_12.diagDIS,
                           CNT_DIAG => #Diagnostic7.ET_200SP.InputsDigital_12.cntDiag);
END_REGION

REGION Network 27
   RUNG wire#powerrail
      GET_DIAG(MODE := #Diagnostic10.ET_200SP.InputsDigital_12.Mode, LADDR := #Diagnostic10.ET_200SP.InputsDigital_12.LADDR, DIAG := #Diagnostic10.ET_200SP.InputsDigital_12.diagDIS, DETAIL :=, RET_VAL => #Diagnostic10.ET_200SP.InputsDigital_12.RetVal, CNT_DIAG => #Diagnostic10.ET_200SP.InputsDigital_12.cntDiag)
   END_RUNG
   // the same network as SCL:
   #Diagnostic10.ET_200SP.InputsDigital_12.RetVal := GET_DIAG(MODE := #Diagnostic10.ET_200SP.InputsDigital_12.Mode,
                           LADDR := #Diagnostic10.ET_200SP.InputsDigital_12.LADDR,
                           DIAG := #Diagnostic10.ET_200SP.InputsDigital_12.diagDIS,
                           CNT_DIAG => #Diagnostic10.ET_200SP.InputsDigital_12.cntDiag);
END_REGION

REGION Network 28
   RUNG wire#powerrail
      GET_DIAG(MODE := #Diagnostic7.ET_200SP.InputsDigital_13.Mode, LADDR := #Diagnostic7.ET_200SP.InputsDigital_13.LADDR, DIAG := #Diagnostic7.ET_200SP.InputsDigital_13.diagDIS, DETAIL :=, RET_VAL => #Diagnostic7.ET_200SP.InputsDigital_13.RetVal, CNT_DIAG => #Diagnostic7.ET_200SP.InputsDigital_13.cntDiag)
   END_RUNG
   // the same network as SCL:
   #Diagnostic7.ET_200SP.InputsDigital_13.RetVal := GET_DIAG(MODE := #Diagnostic7.ET_200SP.InputsDigital_13.Mode,
                           LADDR := #Diagnostic7.ET_200SP.InputsDigital_13.LADDR,
                           DIAG := #Diagnostic7.ET_200SP.InputsDigital_13.diagDIS,
                           CNT_DIAG => #Diagnostic7.ET_200SP.InputsDigital_13.cntDiag);
END_REGION

REGION Network 29
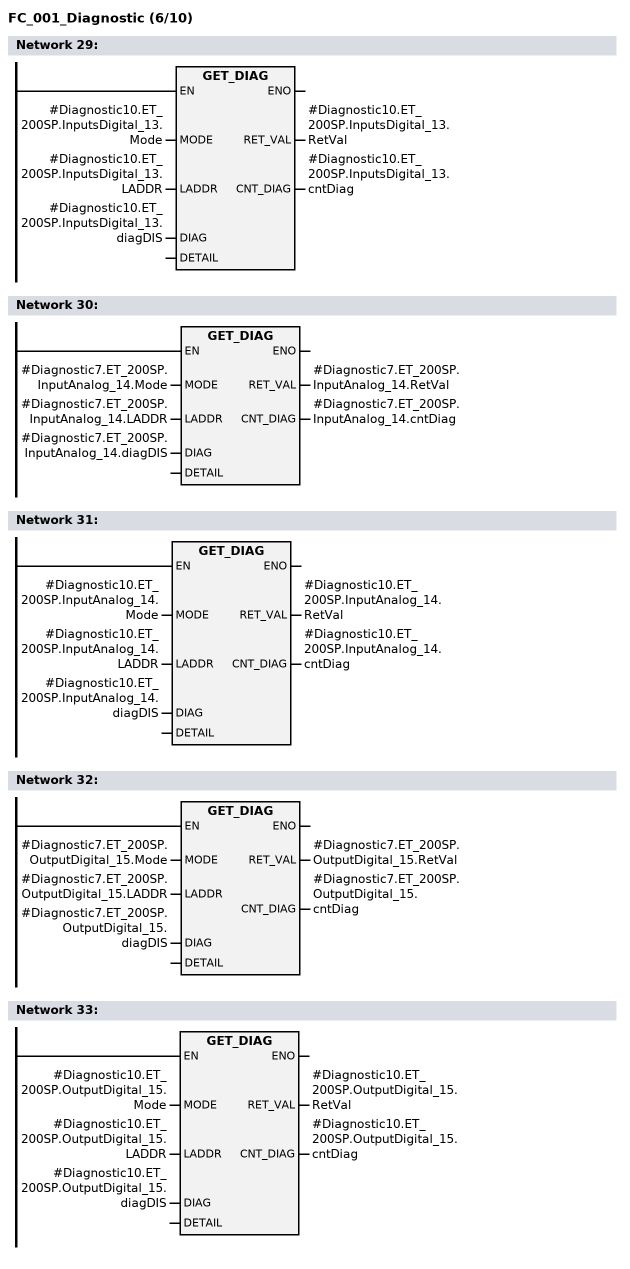
   RUNG wire#powerrail
      GET_DIAG(MODE := #Diagnostic10.ET_200SP.InputsDigital_13.Mode, LADDR := #Diagnostic10.ET_200SP.InputsDigital_13.LADDR, DIAG := #Diagnostic10.ET_200SP.InputsDigital_13.diagDIS, DETAIL :=, RET_VAL => #Diagnostic10.ET_200SP.InputsDigital_13.RetVal, CNT_DIAG => #Diagnostic10.ET_200SP.InputsDigital_13.cntDiag)
   END_RUNG
   // the same network as SCL:
   #Diagnostic10.ET_200SP.InputsDigital_13.RetVal := GET_DIAG(MODE := #Diagnostic10.ET_200SP.InputsDigital_13.Mode,
                           LADDR := #Diagnostic10.ET_200SP.InputsDigital_13.LADDR,
                           DIAG := #Diagnostic10.ET_200SP.InputsDigital_13.diagDIS,
                           CNT_DIAG => #Diagnostic10.ET_200SP.InputsDigital_13.cntDiag);
END_REGION

REGION Network 30
   RUNG wire#powerrail
      GET_DIAG(MODE := #Diagnostic7.ET_200SP.InputAnalog_14.Mode, LADDR := #Diagnostic7.ET_200SP.InputAnalog_14.LADDR, DIAG := #Diagnostic7.ET_200SP.InputAnalog_14.diagDIS, DETAIL :=, RET_VAL => #Diagnostic7.ET_200SP.InputAnalog_14.RetVal, CNT_DIAG => #Diagnostic7.ET_200SP.InputAnalog_14.cntDiag)
   END_RUNG
   // the same network as SCL:
   #Diagnostic7.ET_200SP.InputAnalog_14.RetVal := GET_DIAG(MODE := #Diagnostic7.ET_200SP.InputAnalog_14.Mode,
                           LADDR := #Diagnostic7.ET_200SP.InputAnalog_14.LADDR,
                           DIAG := #Diagnostic7.ET_200SP.InputAnalog_14.diagDIS,
                           CNT_DIAG => #Diagnostic7.ET_200SP.InputAnalog_14.cntDiag);
END_REGION

REGION Network 31
   RUNG wire#powerrail
      GET_DIAG(MODE := #Diagnostic10.ET_200SP.InputAnalog_14.Mode, LADDR := #Diagnostic10.ET_200SP.InputAnalog_14.LADDR, DIAG := #Diagnostic10.ET_200SP.InputAnalog_14.diagDIS, DETAIL :=, RET_VAL => #Diagnostic10.ET_200SP.InputAnalog_14.RetVal, CNT_DIAG => #Diagnostic10.ET_200SP.InputAnalog_14.cntDiag)
   END_RUNG
   // the same network as SCL:
   #Diagnostic10.ET_200SP.InputAnalog_14.RetVal := GET_DIAG(MODE := #Diagnostic10.ET_200SP.InputAnalog_14.Mode,
                           LADDR := #Diagnostic10.ET_200SP.InputAnalog_14.LADDR,
                           DIAG := #Diagnostic10.ET_200SP.InputAnalog_14.diagDIS,
                           CNT_DIAG => #Diagnostic10.ET_200SP.InputAnalog_14.cntDiag);
END_REGION

REGION Network 32
   RUNG wire#powerrail
      GET_DIAG(MODE := #Diagnostic7.ET_200SP.OutputDigital_15.Mode, LADDR := #Diagnostic7.ET_200SP.OutputDigital_15.LADDR, DIAG := #Diagnostic7.ET_200SP.OutputDigital_15.diagDIS, DETAIL :=, RET_VAL => #Diagnostic7.ET_200SP.OutputDigital_15.RetVal, CNT_DIAG => #Diagnostic7.ET_200SP.OutputDigital_15.cntDiag)
   END_RUNG
   // the same network as SCL:
   #Diagnostic7.ET_200SP.OutputDigital_15.RetVal := GET_DIAG(MODE := #Diagnostic7.ET_200SP.OutputDigital_15.Mode,
                           LADDR := #Diagnostic7.ET_200SP.OutputDigital_15.LADDR,
                           DIAG := #Diagnostic7.ET_200SP.OutputDigital_15.diagDIS,
                           CNT_DIAG => #Diagnostic7.ET_200SP.OutputDigital_15.cntDiag);
END_REGION

REGION Network 33
   RUNG wire#powerrail
      GET_DIAG(MODE := #Diagnostic10.ET_200SP.OutputDigital_15.Mode, LADDR := #Diagnostic10.ET_200SP.OutputDigital_15.LADDR, DIAG := #Diagnostic10.ET_200SP.OutputDigital_15.diagDIS, DETAIL :=, RET_VAL => #Diagnostic10.ET_200SP.OutputDigital_15.RetVal, CNT_DIAG => #Diagnostic10.ET_200SP.OutputDigital_15.cntDiag)
   END_RUNG
   // the same network as SCL:
   #Diagnostic10.ET_200SP.OutputDigital_15.RetVal := GET_DIAG(MODE := #Diagnostic10.ET_200SP.OutputDigital_15.Mode,
                           LADDR := #Diagnostic10.ET_200SP.OutputDigital_15.LADDR,
                           DIAG := #Diagnostic10.ET_200SP.OutputDigital_15.diagDIS,
                           CNT_DIAG => #Diagnostic10.ET_200SP.OutputDigital_15.cntDiag);
END_REGION

REGION Network 34
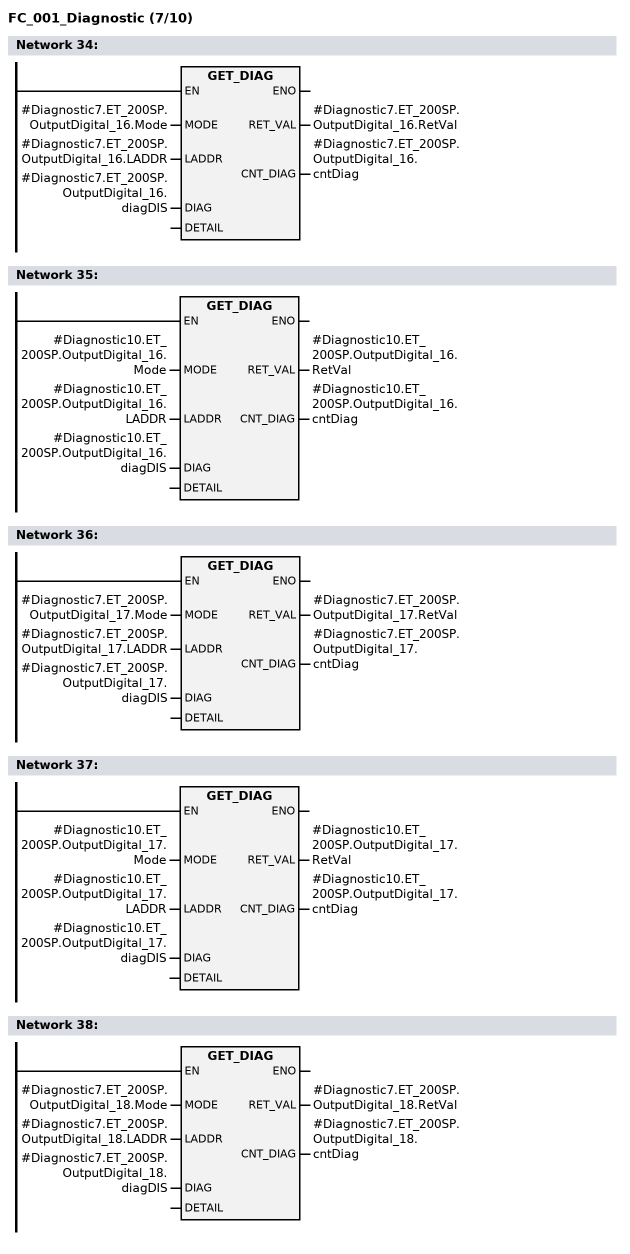
   RUNG wire#powerrail
      GET_DIAG(MODE := #Diagnostic7.ET_200SP.OutputDigital_16.Mode, LADDR := #Diagnostic7.ET_200SP.OutputDigital_16.LADDR, DIAG := #Diagnostic7.ET_200SP.OutputDigital_16.diagDIS, DETAIL :=, RET_VAL => #Diagnostic7.ET_200SP.OutputDigital_16.RetVal, CNT_DIAG => #Diagnostic7.ET_200SP.OutputDigital_16.cntDiag)
   END_RUNG
   // the same network as SCL:
   #Diagnostic7.ET_200SP.OutputDigital_16.RetVal := GET_DIAG(MODE := #Diagnostic7.ET_200SP.OutputDigital_16.Mode,
                           LADDR := #Diagnostic7.ET_200SP.OutputDigital_16.LADDR,
                           DIAG := #Diagnostic7.ET_200SP.OutputDigital_16.diagDIS,
                           CNT_DIAG => #Diagnostic7.ET_200SP.OutputDigital_16.cntDiag);
END_REGION

REGION Network 35
   RUNG wire#powerrail
      GET_DIAG(MODE := #Diagnostic10.ET_200SP.OutputDigital_16.Mode, LADDR := #Diagnostic10.ET_200SP.OutputDigital_16.LADDR, DIAG := #Diagnostic10.ET_200SP.OutputDigital_16.diagDIS, DETAIL :=, RET_VAL => #Diagnostic10.ET_200SP.OutputDigital_16.RetVal, CNT_DIAG => #Diagnostic10.ET_200SP.OutputDigital_16.cntDiag)
   END_RUNG
   // the same network as SCL:
   #Diagnostic10.ET_200SP.OutputDigital_16.RetVal := GET_DIAG(MODE := #Diagnostic10.ET_200SP.OutputDigital_16.Mode,
                           LADDR := #Diagnostic10.ET_200SP.OutputDigital_16.LADDR,
                           DIAG := #Diagnostic10.ET_200SP.OutputDigital_16.diagDIS,
                           CNT_DIAG => #Diagnostic10.ET_200SP.OutputDigital_16.cntDiag);
END_REGION

REGION Network 36
   RUNG wire#powerrail
      GET_DIAG(MODE := #Diagnostic7.ET_200SP.OutputDigital_17.Mode, LADDR := #Diagnostic7.ET_200SP.OutputDigital_17.LADDR, DIAG := #Diagnostic7.ET_200SP.OutputDigital_17.diagDIS, DETAIL :=, RET_VAL => #Diagnostic7.ET_200SP.OutputDigital_17.RetVal, CNT_DIAG => #Diagnostic7.ET_200SP.OutputDigital_17.cntDiag)
   END_RUNG
   // the same network as SCL:
   #Diagnostic7.ET_200SP.OutputDigital_17.RetVal := GET_DIAG(MODE := #Diagnostic7.ET_200SP.OutputDigital_17.Mode,
                           LADDR := #Diagnostic7.ET_200SP.OutputDigital_17.LADDR,
                           DIAG := #Diagnostic7.ET_200SP.OutputDigital_17.diagDIS,
                           CNT_DIAG => #Diagnostic7.ET_200SP.OutputDigital_17.cntDiag);
END_REGION

REGION Network 37
   RUNG wire#powerrail
      GET_DIAG(MODE := #Diagnostic10.ET_200SP.OutputDigital_17.Mode, LADDR := #Diagnostic10.ET_200SP.OutputDigital_17.LADDR, DIAG := #Diagnostic10.ET_200SP.OutputDigital_17.diagDIS, DETAIL :=, RET_VAL => #Diagnostic10.ET_200SP.OutputDigital_17.RetVal, CNT_DIAG => #Diagnostic10.ET_200SP.OutputDigital_17.cntDiag)
   END_RUNG
   // the same network as SCL:
   #Diagnostic10.ET_200SP.OutputDigital_17.RetVal := GET_DIAG(MODE := #Diagnostic10.ET_200SP.OutputDigital_17.Mode,
                           LADDR := #Diagnostic10.ET_200SP.OutputDigital_17.LADDR,
                           DIAG := #Diagnostic10.ET_200SP.OutputDigital_17.diagDIS,
                           CNT_DIAG => #Diagnostic10.ET_200SP.OutputDigital_17.cntDiag);
END_REGION

REGION Network 38
   RUNG wire#powerrail
      GET_DIAG(MODE := #Diagnostic7.ET_200SP.OutputDigital_18.Mode, LADDR := #Diagnostic7.ET_200SP.OutputDigital_18.LADDR, DIAG := #Diagnostic7.ET_200SP.OutputDigital_18.diagDIS, DETAIL :=, RET_VAL => #Diagnostic7.ET_200SP.OutputDigital_18.RetVal, CNT_DIAG => #Diagnostic7.ET_200SP.OutputDigital_18.cntDiag)
   END_RUNG
   // the same network as SCL:
   #Diagnostic7.ET_200SP.OutputDigital_18.RetVal := GET_DIAG(MODE := #Diagnostic7.ET_200SP.OutputDigital_18.Mode,
                           LADDR := #Diagnostic7.ET_200SP.OutputDigital_18.LADDR,
                           DIAG := #Diagnostic7.ET_200SP.OutputDigital_18.diagDIS,
                           CNT_DIAG => #Diagnostic7.ET_200SP.OutputDigital_18.cntDiag);
END_REGION

REGION Network 39
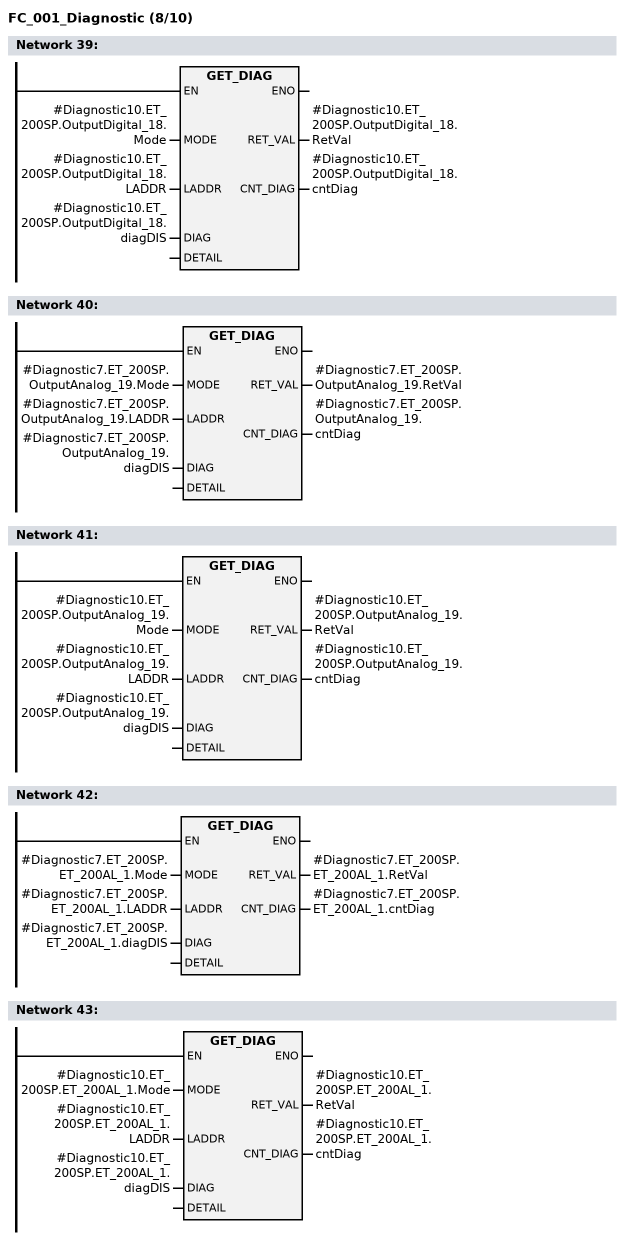
   RUNG wire#powerrail
      GET_DIAG(MODE := #Diagnostic10.ET_200SP.OutputDigital_18.Mode, LADDR := #Diagnostic10.ET_200SP.OutputDigital_18.LADDR, DIAG := #Diagnostic10.ET_200SP.OutputDigital_18.diagDIS, DETAIL :=, RET_VAL => #Diagnostic10.ET_200SP.OutputDigital_18.RetVal, CNT_DIAG => #Diagnostic10.ET_200SP.OutputDigital_18.cntDiag)
   END_RUNG
   // the same network as SCL:
   #Diagnostic10.ET_200SP.OutputDigital_18.RetVal := GET_DIAG(MODE := #Diagnostic10.ET_200SP.OutputDigital_18.Mode,
                           LADDR := #Diagnostic10.ET_200SP.OutputDigital_18.LADDR,
                           DIAG := #Diagnostic10.ET_200SP.OutputDigital_18.diagDIS,
                           CNT_DIAG => #Diagnostic10.ET_200SP.OutputDigital_18.cntDiag);
END_REGION

REGION Network 40
   RUNG wire#powerrail
      GET_DIAG(MODE := #Diagnostic7.ET_200SP.OutputAnalog_19.Mode, LADDR := #Diagnostic7.ET_200SP.OutputAnalog_19.LADDR, DIAG := #Diagnostic7.ET_200SP.OutputAnalog_19.diagDIS, DETAIL :=, RET_VAL => #Diagnostic7.ET_200SP.OutputAnalog_19.RetVal, CNT_DIAG => #Diagnostic7.ET_200SP.OutputAnalog_19.cntDiag)
   END_RUNG
   // the same network as SCL:
   #Diagnostic7.ET_200SP.OutputAnalog_19.RetVal := GET_DIAG(MODE := #Diagnostic7.ET_200SP.OutputAnalog_19.Mode,
                           LADDR := #Diagnostic7.ET_200SP.OutputAnalog_19.LADDR,
                           DIAG := #Diagnostic7.ET_200SP.OutputAnalog_19.diagDIS,
                           CNT_DIAG => #Diagnostic7.ET_200SP.OutputAnalog_19.cntDiag);
END_REGION

REGION Network 41
   RUNG wire#powerrail
      GET_DIAG(MODE := #Diagnostic10.ET_200SP.OutputAnalog_19.Mode, LADDR := #Diagnostic10.ET_200SP.OutputAnalog_19.LADDR, DIAG := #Diagnostic10.ET_200SP.OutputAnalog_19.diagDIS, DETAIL :=, RET_VAL => #Diagnostic10.ET_200SP.OutputAnalog_19.RetVal, CNT_DIAG => #Diagnostic10.ET_200SP.OutputAnalog_19.cntDiag)
   END_RUNG
   // the same network as SCL:
   #Diagnostic10.ET_200SP.OutputAnalog_19.RetVal := GET_DIAG(MODE := #Diagnostic10.ET_200SP.OutputAnalog_19.Mode,
                           LADDR := #Diagnostic10.ET_200SP.OutputAnalog_19.LADDR,
                           DIAG := #Diagnostic10.ET_200SP.OutputAnalog_19.diagDIS,
                           CNT_DIAG => #Diagnostic10.ET_200SP.OutputAnalog_19.cntDiag);
END_REGION

REGION Network 42
   RUNG wire#powerrail
      GET_DIAG(MODE := #Diagnostic7.ET_200SP.ET_200AL_1.Mode, LADDR := #Diagnostic7.ET_200SP.ET_200AL_1.LADDR, DIAG := #Diagnostic7.ET_200SP.ET_200AL_1.diagDIS, DETAIL :=, RET_VAL => #Diagnostic7.ET_200SP.ET_200AL_1.RetVal, CNT_DIAG => #Diagnostic7.ET_200SP.ET_200AL_1.cntDiag)
   END_RUNG
   // the same network as SCL:
   #Diagnostic7.ET_200SP.ET_200AL_1.RetVal := GET_DIAG(MODE := #Diagnostic7.ET_200SP.ET_200AL_1.Mode,
                           LADDR := #Diagnostic7.ET_200SP.ET_200AL_1.LADDR,
                           DIAG := #Diagnostic7.ET_200SP.ET_200AL_1.diagDIS,
                           CNT_DIAG => #Diagnostic7.ET_200SP.ET_200AL_1.cntDiag);
END_REGION

REGION Network 43
   RUNG wire#powerrail
      GET_DIAG(MODE := #Diagnostic10.ET_200SP.ET_200AL_1.Mode, LADDR := #Diagnostic10.ET_200SP.ET_200AL_1.LADDR, DIAG := #Diagnostic10.ET_200SP.ET_200AL_1.diagDIS, DETAIL :=, RET_VAL => #Diagnostic10.ET_200SP.ET_200AL_1.RetVal, CNT_DIAG => #Diagnostic10.ET_200SP.ET_200AL_1.cntDiag)
   END_RUNG
   // the same network as SCL:
   #Diagnostic10.ET_200SP.ET_200AL_1.RetVal := GET_DIAG(MODE := #Diagnostic10.ET_200SP.ET_200AL_1.Mode,
                           LADDR := #Diagnostic10.ET_200SP.ET_200AL_1.LADDR,
                           DIAG := #Diagnostic10.ET_200SP.ET_200AL_1.diagDIS,
                           CNT_DIAG => #Diagnostic10.ET_200SP.ET_200AL_1.cntDiag);
END_REGION

REGION Network 44
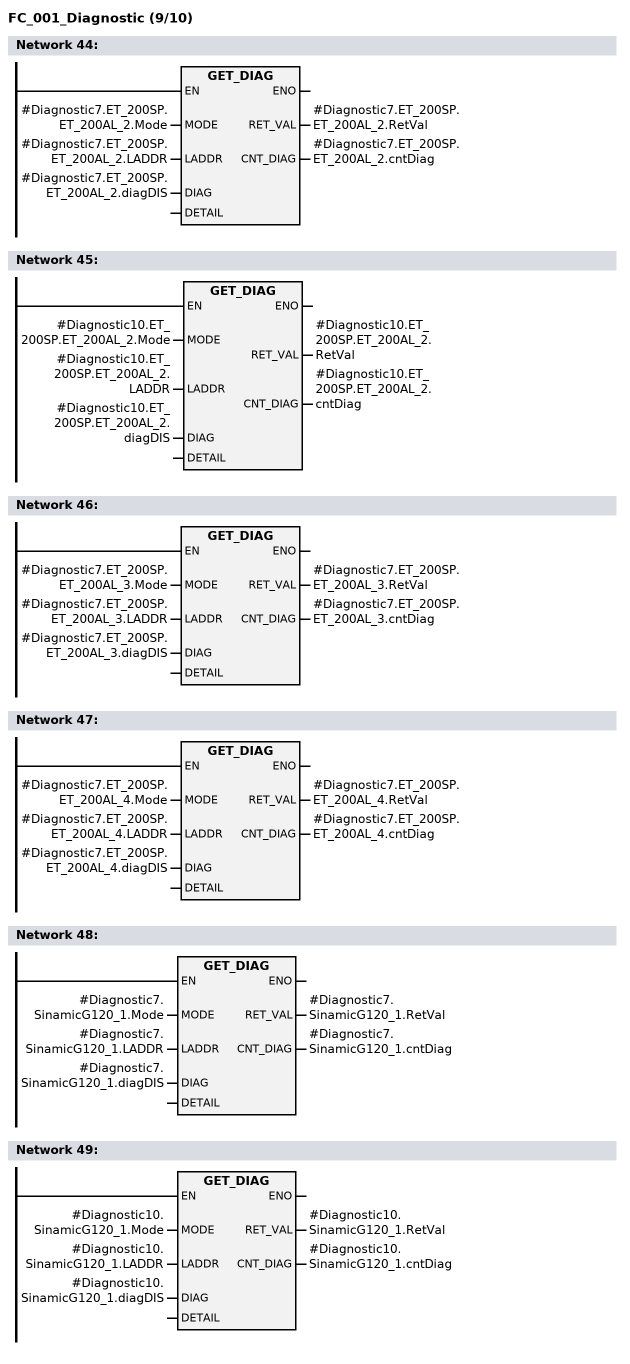
   RUNG wire#powerrail
      GET_DIAG(MODE := #Diagnostic7.ET_200SP.ET_200AL_2.Mode, LADDR := #Diagnostic7.ET_200SP.ET_200AL_2.LADDR, DIAG := #Diagnostic7.ET_200SP.ET_200AL_2.diagDIS, DETAIL :=, RET_VAL => #Diagnostic7.ET_200SP.ET_200AL_2.RetVal, CNT_DIAG => #Diagnostic7.ET_200SP.ET_200AL_2.cntDiag)
   END_RUNG
   // the same network as SCL:
   #Diagnostic7.ET_200SP.ET_200AL_2.RetVal := GET_DIAG(MODE := #Diagnostic7.ET_200SP.ET_200AL_2.Mode,
                           LADDR := #Diagnostic7.ET_200SP.ET_200AL_2.LADDR,
                           DIAG := #Diagnostic7.ET_200SP.ET_200AL_2.diagDIS,
                           CNT_DIAG => #Diagnostic7.ET_200SP.ET_200AL_2.cntDiag);
END_REGION

REGION Network 45
   RUNG wire#powerrail
      GET_DIAG(MODE := #Diagnostic10.ET_200SP.ET_200AL_2.Mode, LADDR := #Diagnostic10.ET_200SP.ET_200AL_2.LADDR, DIAG := #Diagnostic10.ET_200SP.ET_200AL_2.diagDIS, DETAIL :=, RET_VAL => #Diagnostic10.ET_200SP.ET_200AL_2.RetVal, CNT_DIAG => #Diagnostic10.ET_200SP.ET_200AL_2.cntDiag)
   END_RUNG
   // the same network as SCL:
   #Diagnostic10.ET_200SP.ET_200AL_2.RetVal := GET_DIAG(MODE := #Diagnostic10.ET_200SP.ET_200AL_2.Mode,
                           LADDR := #Diagnostic10.ET_200SP.ET_200AL_2.LADDR,
                           DIAG := #Diagnostic10.ET_200SP.ET_200AL_2.diagDIS,
                           CNT_DIAG => #Diagnostic10.ET_200SP.ET_200AL_2.cntDiag);
END_REGION

REGION Network 46
   RUNG wire#powerrail
      GET_DIAG(MODE := #Diagnostic7.ET_200SP.ET_200AL_3.Mode, LADDR := #Diagnostic7.ET_200SP.ET_200AL_3.LADDR, DIAG := #Diagnostic7.ET_200SP.ET_200AL_3.diagDIS, DETAIL :=, RET_VAL => #Diagnostic7.ET_200SP.ET_200AL_3.RetVal, CNT_DIAG => #Diagnostic7.ET_200SP.ET_200AL_3.cntDiag)
   END_RUNG
   // the same network as SCL:
   #Diagnostic7.ET_200SP.ET_200AL_3.RetVal := GET_DIAG(MODE := #Diagnostic7.ET_200SP.ET_200AL_3.Mode,
                           LADDR := #Diagnostic7.ET_200SP.ET_200AL_3.LADDR,
                           DIAG := #Diagnostic7.ET_200SP.ET_200AL_3.diagDIS,
                           CNT_DIAG => #Diagnostic7.ET_200SP.ET_200AL_3.cntDiag);
END_REGION

REGION Network 47
   RUNG wire#powerrail
      GET_DIAG(MODE := #Diagnostic7.ET_200SP.ET_200AL_4.Mode, LADDR := #Diagnostic7.ET_200SP.ET_200AL_4.LADDR, DIAG := #Diagnostic7.ET_200SP.ET_200AL_4.diagDIS, DETAIL :=, RET_VAL => #Diagnostic7.ET_200SP.ET_200AL_4.RetVal, CNT_DIAG => #Diagnostic7.ET_200SP.ET_200AL_4.cntDiag)
   END_RUNG
   // the same network as SCL:
   #Diagnostic7.ET_200SP.ET_200AL_4.RetVal := GET_DIAG(MODE := #Diagnostic7.ET_200SP.ET_200AL_4.Mode,
                           LADDR := #Diagnostic7.ET_200SP.ET_200AL_4.LADDR,
                           DIAG := #Diagnostic7.ET_200SP.ET_200AL_4.diagDIS,
                           CNT_DIAG => #Diagnostic7.ET_200SP.ET_200AL_4.cntDiag);
END_REGION

REGION Network 48
   RUNG wire#powerrail
      GET_DIAG(MODE := #Diagnostic7.SinamicG120_1.Mode, LADDR := #Diagnostic7.SinamicG120_1.LADDR, DIAG := #Diagnostic7.SinamicG120_1.diagDIS, DETAIL :=, RET_VAL => #Diagnostic7.SinamicG120_1.RetVal, CNT_DIAG => #Diagnostic7.SinamicG120_1.cntDiag)
   END_RUNG
   // the same network as SCL:
   #Diagnostic7.SinamicG120_1.RetVal := GET_DIAG(MODE := #Diagnostic7.SinamicG120_1.Mode,
                           LADDR := #Diagnostic7.SinamicG120_1.LADDR,
                           DIAG := #Diagnostic7.SinamicG120_1.diagDIS,
                           CNT_DIAG => #Diagnostic7.SinamicG120_1.cntDiag);
END_REGION

REGION Network 49
   RUNG wire#powerrail
      GET_DIAG(MODE := #Diagnostic10.SinamicG120_1.Mode, LADDR := #Diagnostic10.SinamicG120_1.LADDR, DIAG := #Diagnostic10.SinamicG120_1.diagDIS, DETAIL :=, RET_VAL => #Diagnostic10.SinamicG120_1.RetVal, CNT_DIAG => #Diagnostic10.SinamicG120_1.cntDiag)
   END_RUNG
   // the same network as SCL:
   #Diagnostic10.SinamicG120_1.RetVal := GET_DIAG(MODE := #Diagnostic10.SinamicG120_1.Mode,
                           LADDR := #Diagnostic10.SinamicG120_1.LADDR,
                           DIAG := #Diagnostic10.SinamicG120_1.diagDIS,
                           CNT_DIAG => #Diagnostic10.SinamicG120_1.cntDiag);
END_REGION

REGION Network 50
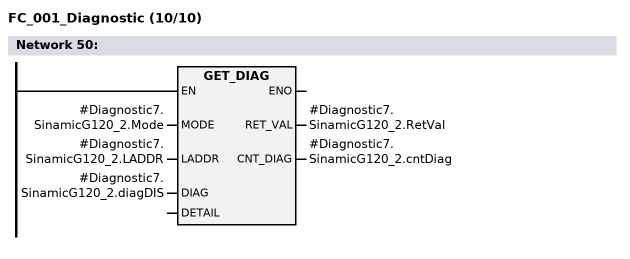
   RUNG wire#powerrail
      GET_DIAG(MODE := #Diagnostic7.SinamicG120_2.Mode, LADDR := #Diagnostic7.SinamicG120_2.LADDR, DIAG := #Diagnostic7.SinamicG120_2.diagDIS, DETAIL :=, RET_VAL => #Diagnostic7.SinamicG120_2.RetVal, CNT_DIAG => #Diagnostic7.SinamicG120_2.cntDiag)
   END_RUNG
   // the same network as SCL:
   #Diagnostic7.SinamicG120_2.RetVal := GET_DIAG(MODE := #Diagnostic7.SinamicG120_2.Mode,
                           LADDR := #Diagnostic7.SinamicG120_2.LADDR,
                           DIAG := #Diagnostic7.SinamicG120_2.diagDIS,
                           CNT_DIAG => #Diagnostic7.SinamicG120_2.cntDiag);
END_REGION

REGION Network 51 (SCL)
   // Diagnostyka dla szafy 1
   #Diagnostic7.DiagnosticOK := #Diagnostic7.ET_200SP.HeadModule_0.diagDIS.OwnState = 0 AND
   #Diagnostic7.ET_200SP.BusAdapter_1.diagDIS.OwnState = 0 AND #Diagnostic7.ET_200SP.InputSafety_2.diagDIS.OwnState = 0 AND
   #Diagnostic7.ET_200SP.InputSafety_3.diagDIS.OwnState = 0 AND #Diagnostic7.ET_200SP.InputSafety_4.diagDIS.OwnState = 0 AND
   #Diagnostic7.ET_200SP.InputSafety_5.diagDIS.OwnState = 0 AND #Diagnostic7.ET_200SP.OutputSafety_7.diagDIS.OwnState = 0 AND
   #Diagnostic7.ET_200SP.RelaySafety_9.diagDIS.OwnState = 0 AND #Diagnostic7.ET_200SP.InputSafety_6.diagDIS.OwnState = 0 AND
   #Diagnostic7.ET_200SP.RelaySafety_10.diagDIS.OwnState = 0 AND #Diagnostic7.ET_200SP.InputsDigital_11.diagDIS.OwnState = 0 AND
   #Diagnostic7.ET_200SP.InputsDigital_12.diagDIS.OwnState = 0 AND #Diagnostic7.ET_200SP.InputsDigital_13.diagDIS.OwnState = 0 AND
   #Diagnostic7.ET_200SP.InputAnalog_14.diagDIS.OwnState = 0 AND #Diagnostic7.ET_200SP.OutputDigital_15.diagDIS.OwnState = 0 AND
   #Diagnostic7.ET_200SP.OutputDigital_16.diagDIS.OwnState = 0 AND #Diagnostic7.ET_200SP.OutputDigital_17.diagDIS.OwnState = 0 AND
   #Diagnostic7.ET_200SP.OutputDigital_18.diagDIS.OwnState = 0 AND #Diagnostic7.ET_200SP.OutputAnalog_19.diagDIS.OwnState = 0 AND
   #Diagnostic7.ET_200SP.ET_200AL_1.diagDIS.OwnState = 0 AND #Diagnostic7.ET_200SP.ET_200AL_2.diagDIS.OwnState = 0 AND
   #Diagnostic7.ET_200SP.ET_200AL_3.diagDIS.OwnState = 0 AND #Diagnostic7.ET_200SP.ET_200AL_4.diagDIS.OwnState = 0 AND
   #Diagnostic7.SinamicG120_1.diagDIS.OwnState = 0 AND #Diagnostic7.SinamicG120_2.diagDIS.OwnState = 0;
END_REGION

REGION Network 52 (SCL)
   //DIAGNOSTYKA 10 
   #Diagnostic10.DiagnosticOK := #Diagnostic10.ET_200SP.HeadModule_0.diagDIS.OwnState = 0 AND
   #Diagnostic10.ET_200SP.BusAdapter_1.diagDIS.OwnState = 0 AND #Diagnostic10.ET_200SP.InputSafety_2.diagDIS.OwnState = 0 AND
   #Diagnostic10.ET_200SP.InputSafety_3.diagDIS.OwnState = 0 AND #Diagnostic10.ET_200SP.InputSafety_4.diagDIS.OwnState = 0 AND
   #Diagnostic10.ET_200SP.InputSafety_5.diagDIS.OwnState = 0 AND #Diagnostic10.ET_200SP.OutputSafety_7.diagDIS.OwnState = 0 AND
   #Diagnostic10.ET_200SP.RelaySafety_9.diagDIS.OwnState = 0 AND #Diagnostic10.ET_200SP.InputSafety_6.diagDIS.OwnState = 0 AND
   #Diagnostic10.ET_200SP.RelaySafety_10.diagDIS.OwnState = 0 AND #Diagnostic10.ET_200SP.InputsDigital_11.diagDIS.OwnState = 0 AND
   #Diagnostic10.ET_200SP.InputsDigital_12.diagDIS.OwnState = 0 AND #Diagnostic10.ET_200SP.InputsDigital_13.diagDIS.OwnState = 0 AND
   #Diagnostic10.ET_200SP.InputAnalog_14.diagDIS.OwnState = 0 AND #Diagnostic10.ET_200SP.OutputDigital_15.diagDIS.OwnState = 0 AND
   #Diagnostic10.ET_200SP.OutputDigital_16.diagDIS.OwnState = 0 AND #Diagnostic10.ET_200SP.OutputDigital_17.diagDIS.OwnState = 0 AND
   #Diagnostic10.ET_200SP.OutputDigital_18.diagDIS.OwnState = 0 AND #Diagnostic10.ET_200SP.OutputAnalog_19.diagDIS.OwnState = 0 AND
   #Diagnostic10.ET_200SP.ET_200AL_1.diagDIS.OwnState = 0 AND #Diagnostic10.ET_200SP.ET_200AL_2.diagDIS.OwnState = 0 AND
   #Diagnostic10.SinamicG120_1.diagDIS.OwnState = 0;
END_REGION
END_FUNCTION
